// TIA Portal V17 export
// export: Created 2025-06-26T06:49:28.1855995Z, ExportSetting WithDefaults, DisplayName Totally Integrated Automation Portal, DisplayVersion V17 Update 8, DisplayName TIA Portal Openness, DisplayVersion V17 Update 8, DisplayName TIA Portal Version Control Interface, DisplayVersion V17, DisplayName STEP 7 Professional, DisplayVersion V17 Update 8, DisplayName STEP 7 Safety, DisplayVersion V17 Update 6, DisplayName WinCC Advanced, DisplayVersion V17 Update 8
TYPE "stCalcSelect"
// stored: IsFailsafeCompliant false
   STRUCT
      nMode : USInt;   // Requested mode (0 = none, 1 = A, 2 = B, 3 = MIN, 4 = MAX, 5 = AVG)
      nActualMode : USInt;   // Actual mode (differs from nMode if bWarning is true)
      bError : Bool;   // 1 = not able to emit any output value, 0 = value ok
      bWarning : Bool;   // 1 = not able to emit requested value, 0 = value ok
   END_STRUCT;
END_TYPE
